FUNCTION_BLOCK FINAL Action_Person_ IMPLEMENTS I_Action

METHOD Perform
VAR_INPUT
    performCaseNumber : INT;
END_VAR
VAR_IN_OUT
	item : POINTER TO Object;
END_VAR
CASE performCaseNumber OF
    1 :
    GVL.CastHelper.ObjectToPerson(item)^.SetAge(50);
    2 :
    GVL.CastHelper.ObjectToPerson(item)^.SetName('Sylvia');
ELSE
    RETURN;
END_CASE
END_METHOD

END_FUNCTION_BLOCK

(* stored: Version 1.1.0.1, ProductVersion 3.1.4024.6
   POU Action_Person_: Id {b5be6651-38ea-4258-9eec-f3671df0c0ae}, SpecialFunc None
   Method Perform: Id {a2abe9cf-f46d-4c8a-b5ae-074ef44d8a54} *)
